// TwinCAT 3 PLC project LoadCellReader
// ProgramVersion: 3.1.4024.0
// libraries:
//   Tc2_Standard, * (Beckhoff Automation GmbH)
//   Tc2_System, * (Beckhoff Automation GmbH)
//   Tc3_Module, * (Beckhoff Automation GmbH)
// project tree:
//   GVLs/ GVL_Receive.TcGVL, GVL_Transmit.TcGVL
//   / PlcTask.TcTTO
//   POUs/FunctionBlocks/ EvaluateAllOffsets.TcPOU
//   POUs/Functions/ EvaluateOffset.TcPOU, ScaleVoltage.TcPOU
//   POUs/ MAIN.TcPOU

CONFIGURATION LoadCellReader
    RESOURCE PLC ON TwinCAT3
        TASK PlcTask(INTERVAL := T#1ms, PRIORITY := 11);
        PROGRAM MAIN WITH PlcTask : MAIN;
    END_RESOURCE
END_CONFIGURATION

// ---- GVLs/GVL_Receive.TcGVL
{attribute 'qualified_only'}

// This Global variable List holds all Globals received from the control PC over ADS and raw voltages (binary) from the PLC
VAR_GLOBAL
	
	bTransmitVoltages AT %I* : BOOL;				// to recieve from control PC whether to transmit the voltages to the control PC
	bCalculateOffset AT %I* : BOOL;					// Command to recalculate offset
	
	iRawAI1 AT %I* : INT;							// Raw voltage in binary from the PLC AI1
	iRawAI2 AT %I* : INT;							// Raw voltage in binary from the PLC AI2
	iRawAI3 AT %I* : INT;							// Raw voltage in binary from the PLC AI3
	iRawAI4 AT %I* : INT;							// Raw voltage in binary from the PLC AI4
	iRawAI5 AT %I* : INT;							// Raw voltage in binary from the PLC AI5
	iRawAI6 AT %I* : INT;							// Raw voltage in binary from the PLC AI6
	
	fOffsetAI1 AT %I* : REAL;						// Voltage Offset calculated from Raw AI
	fOffsetAI2 AT %I* : REAL;						// Voltage Offset calculated from Raw AI
	fOffsetAI3 AT %I* : REAL;						// Voltage Offset calculated from Raw AI
	fOffsetAI4 AT %I* : REAL;						// Voltage Offset calculated from Raw AI
	fOffsetAI5 AT %I* : REAL;						// Voltage Offset calculated from Raw AI
	fOffsetAI6 AT %I* : REAL;						// Voltage Offset calculated from Raw AI
	
END_VAR

// ---- GVLs/GVL_Transmit.TcGVL
{attribute 'qualified_only'}

// This Global variable List holds all Globals transmitted to the control PC over ADS
VAR_GLOBAL
	
	fTransmitAI1 AT %Q* : REAL;			// to transmit the voltage at AI 1
	fTransmitAI2 AT %Q* : REAL;			// to transmit the voltage at AI 2
	fTransmitAI3 AT %Q* : REAL;			// to transmit the voltage at AI 3
	fTransmitAI4 AT %Q* : REAL;			// to transmit the voltage at AI 4
	fTransmitAI5 AT %Q* : REAL;			// to transmit the voltage at AI 5
	fTransmitAI6 AT %Q* : REAL;			// to transmit the voltage at AI 6
	
END_VAR

// ---- POUs/MAIN.TcPOU
PROGRAM MAIN
VAR

	bInit : BOOL := TRUE;	
	fbEvaluateOffsets: EvaluateAllOffsets; // Instance of EvaluateAllOffsets
END_VAR

(*
		This project reads the voltages from the Loadcell and transmits the data across ADS.
		
		1. Connect variables to hardware
		2. Read the voltage of each channel
		3. Convert from binary to float
		4. transmit across ADS

*)

// Initiliase the offsets and transmission variables
IF (bInit) THEN
	
	// Call the fucntion block that evaluates all the offsets
	fbEvaluateOffsets();
	
	GVL_Transmit.fTransmitAI1 := 0.0;
	GVL_Transmit.fTransmitAI2 := 0.0;
	GVL_Transmit.fTransmitAI3 := 0.0;
	GVL_Transmit.fTransmitAI4 := 0.0;
	GVL_Transmit.fTransmitAI5 := 0.0;
	GVL_Transmit.fTransmitAI6 := 0.0;
	
	bInit := FALSE;

END_IF

// Check whether to recalculate offsets
IF (GVL_Receive.bCalculateOffset) THEN
	// Call the fucntion block that evaluates all the offsets
	fbEvaluateOffsets();
	
	GVL_Receive.bCalculateOffset := FALSE;

END_IF

// If ready to recieve, scale and transmit the data
IF (GVL_Receive.bTransmitVoltages) THEN

	// Update the Globals which will be transmitted to the control PC
	GVL_Transmit.fTransmitAI1 := (ScaleVoltage(GVL_Receive.iRawAI1)) + GVL_Receive.fOffsetAI1;
	GVL_Transmit.fTransmitAI2 := (ScaleVoltage(GVL_Receive.iRawAI2)) + GVL_Receive.fOffsetAI2;
	GVL_Transmit.fTransmitAI3 := (ScaleVoltage(GVL_Receive.iRawAI3)) + GVL_Receive.fOffsetAI3;
	GVL_Transmit.fTransmitAI4 := (ScaleVoltage(GVL_Receive.iRawAI4)) + GVL_Receive.fOffsetAI4;
	GVL_Transmit.fTransmitAI5 := (ScaleVoltage(GVL_Receive.iRawAI5)) + GVL_Receive.fOffsetAI5;
	GVL_Transmit.fTransmitAI6 := (ScaleVoltage(GVL_Receive.iRawAI6)) + GVL_Receive.fOffsetAI6;
	
ELSE
	
	// Not ready to transmit, only write 0.0 to the Transmit GVLs
	GVL_Transmit.fTransmitAI1 := 0.0;
	GVL_Transmit.fTransmitAI2 := 0.0;
	GVL_Transmit.fTransmitAI3 := 0.0;
	GVL_Transmit.fTransmitAI4 := 0.0;
	GVL_Transmit.fTransmitAI5 := 0.0;
	GVL_Transmit.fTransmitAI6 := 0.0;
	
END_IF

END_PROGRAM

// ---- POUs/FunctionBlocks/EvaluateAllOffsets.TcPOU
FUNCTION_BLOCK EvaluateAllOffsets
VAR_INPUT
END_VAR
VAR_OUTPUT
END_VAR
VAR
END_VAR

	
// This function block calculates all the offsets

GVL_Receive.fOffsetAI1 := EvaluateOffset(ScaleVoltage(GVL_Receive.iRawAI1));
GVL_Receive.fOffsetAI2 := EvaluateOffset(ScaleVoltage(GVL_Receive.iRawAI2));
GVL_Receive.fOffsetAI3 := EvaluateOffset(ScaleVoltage(GVL_Receive.iRawAI3));
GVL_Receive.fOffsetAI4 := EvaluateOffset(ScaleVoltage(GVL_Receive.iRawAI4));
GVL_Receive.fOffsetAI5 := EvaluateOffset(ScaleVoltage(GVL_Receive.iRawAI5));
GVL_Receive.fOffsetAI6 := EvaluateOffset(ScaleVoltage(GVL_Receive.iRawAI6));

END_FUNCTION_BLOCK

// ---- POUs/Functions/EvaluateOffset.TcPOU
FUNCTION EvaluateOffset : REAL
VAR_INPUT
	fRaw : REAL;				// Voltage reading (binary) from HW
END_VAR
VAR
END_VAR

EvaluateOffset := 0.0 - fRaw;

END_FUNCTION

// ---- POUs/Functions/ScaleVoltage.TcPOU
FUNCTION ScaleVoltage : REAL
// Straight Lie Interpolation for Scaling Analog Signals.
// Targeted specifically for +/- 10V at 16 bit resolution
VAR_INPUT
	iRawInput : INT;				// Voltage reading (binary) from HW
END_VAR
VAR
	iResolution : INT := 32767;		// resolution of the ADC (16 bit corresponding to 32767)
	fVoltageLow : REAL := -10.0;	// Lower Limit of the voltage range
	fVoltageHigh : REAL := 10.0;	// Upper Limit of the voltage range
END_VAR

// Vin = 0bRawIn/0bResolution * VoltageMeasurementRange + Offset

ScaleVoltage := (INT_TO_REAL(iRawInput) / INT_TO_REAL(iResolution)) * (fVoltageHigh - fVoltageLow);// - fVoltageHigh;

END_FUNCTION
